(* CODESYS project M241_ILE_writeCSV.project
   Title: M241-ILS2K
   Version: 0.0.0.0
   Author: Philippe

Project tree, tasks and I/O mapping:
  MyController : TM241CE40R, Schneider Electric, order no. TM241CE40R, version 5.1.9.44
    application Application
      libraries: Integrated Lexium Library, 3.2.1.0 (Schneider Electric); FileFormatUtility, 1.5.15.0 (Schneider Electric)
      task MAST (cyclic, interval 20 ms, priority 15, watchdog 100 ms x 1) calls UPDATE_COMMAND, MAIN_SFC, CONSIGNE_VITESSE, ILE_functionblocks
      task Initialisation_IO (event, event StartApp, priority 1) calls nothing
      global variables GVL
      visualisation Visualization
      program ILE_functionblocks [FBD]
      program MAIN_SFC [SFC]
      visualisation Visualization_1
      program UPDATE_COMMAND [SFC]: WRITE_TABLE
      program CONSIGNE_VITESSE [ST]
    DI : Digital Inputs, Schneider Electric, version 5.1.9.44
        input  idwDI_IDW0 : DWORD  // IDW0
        input  ibDI_IB1 : BYTE  // IB1
    DQ : Digital Outputs, Schneider Electric, version 5.1.9.44
        output qwDQ_QW0 : WORD  // QW0
        output qbDQ_QB1 : BYTE  // QB1
    Counters : Counters, Schneider Electric, version 5.1.9.44
    Pulse_Generators : Pulse Generators, Schneider Electric, version 5.1.9.44
    Cartridge_1 : Cartridge, Schneider Electric, version 5.1.9.44
    Cartridge_2 : Cartridge, Schneider Electric, version 5.1.9.44
    IO_Bus : IO bus - TM3, Schneider Electric, version 5.1.9.44
    COM_Bus : COM bus, Schneider Electric, version 5.1.9.44
    Ethernet_1 : Ethernet Network, Schneider Electric, version 5.1.9.44
        settings: IPAddress = [192, 168, 100, 200]; SubnetMask = [255, 255, 255, 0]; GatewayAddress = [192, 168, 100, 254]; WebServer = TRUE; FTP Server = TRUE; SoMachine Protocol = TRUE; Modbus Server = TRUE; NetManage Protocol = TRUE; SNMP protocol = TRUE; Enable Routing = FALSE; WebVisu protocol = TRUE; DHCP Server Active = TRUE; Secured Web Server = TRUE
      Gestionnaire_Ethernet_Industriel : Industrial Ethernet Manager, Schneider Electric, version 1.0.12.40
          settings: BinaryFileSize = 586; Dhcps Host 0.Client Mac Address = [16#00, 16#80, 16#F4, 16#7B, 16#28, 16#E1]; Dhcps Host 0.Client Device Name = 'Lexium-ILx-002'; Dhcps Host 0.Client IP Address = [192, 168, 100, 159]; Dhcps Host 0.Network Mask = [255, 255, 255, 0]; Dhcps Host 0.Default Gateway = [192, 168, 100, 200]; Dhcps Host 2.Client Mac Address = [16#0, 16#0, 16#0, 16#0, 16#0]; Dhcps Host 3.Client Mac Address = [16#0, 16#0, 16#0, 16#0, 16#0]; Dhcps Host 4.Client Mac Address = [16#0, 16#0, 16#0, 16#0, 16#0]; Dhcps Host 5.Client Mac Address = [16#0, 16#0, 16#0, 16#0, 16#0]; Dhcps Host 6.Client Mac Address = [16#0, 16#0, 16#0, 16#0, 16#0]; Dhcps Host 7.Client Mac Address = [16#0, 16#0, 16#0, 16#0, 16#0]; Dhcps Host 8.Client Mac Address = [16#0, 16#0, 16#0, 16#0, 16#0]; Dhcps Host 9.Client Mac Address = [16#0, 16#0, 16#0, 16#0, 16#0]; Dhcps Host 10.Client Mac Address = [16#0, 16#0, 16#0, 16#0, 16#0]; Dhcps Host 11.Client Mac Address = [16#0, 16#0, 16#0, 16#0, 16#0]; Dhcps Host 12.Client Mac Address = [16#0, 16#0, 16#0, 16#0, 16#0]; Dhcps Host 13.Client Mac Address = [16#0, 16#0, 16#0, 16#0, 16#0]; Dhcps Host 14.Client Mac Address = [16#0, 16#0, 16#0, 16#0, 16#0]; Dhcps Host 15.Client Mac Address = [16#0, 16#0, 16#0, 16#0, 16#0]; Dhcps Host 16.Client Mac Address = [16#0, 16#0, 16#0, 16#0, 16#0]; Dhcps Host 17.Client Mac Address = [16#0, 16#0, 16#0, 16#0, 16#0]; Dhcps Host 18.Client Mac Address = [16#0, 16#0, 16#0, 16#0, 16#0]; Dhcps Host 19.Client Mac Address = [16#0, 16#0, 16#0, 16#0, 16#0]; Dhcps Host 20.Client Mac Address = [16#0, 16#0, 16#0, 16#0, 16#0]; Dhcps Host 21.Client Mac Address = [16#0, 16#0, 16#0, 16#0, 16#0]; Dhcps Host 22.Client Mac Address = [16#0, 16#0, 16#0, 16#0, 16#0]; Dhcps Host 23.Client Mac Address = [16#0, 16#0, 16#0, 16#0, 16#0]; Dhcps Host 24.Client Mac Address = [16#0, 16#0, 16#0, 16#0, 16#0]; Dhcps Host 25.Client Mac Address = [16#0, 16#0, 16#0, 16#0, 16#0]; Dhcps Host 26.Client Mac Address = [16#0, 16#0, 16#0, 16#0, 16#0]; Dhcps Host 27.Client Mac Address = [16#0, 16#0, 16#0, 16#0, 16#0]; Dhcps Host 28.Client Mac Address = [16#0, 16#0, 16#0, 16#0, 16#0]; Dhcps Host 29.Client Mac Address = [16#0, 16#0, 16#0, 16#0, 16#0]; Dhcps Host 30.Client Mac Address = [16#0, 16#0, 16#0, 16#0, 16#0]; Dhcps Host 31.Client Mac Address = [16#0, 16#0, 16#0, 16#0, 16#0]; Dhcps Host 32.Client Mac Address = [16#0, 16#0, 16#0, 16#0, 16#0]; Dhcps Host 33.Client Mac Address = [16#0, 16#0, 16#0, 16#0, 16#0]; Dhcps Host 34.Client Mac Address = [16#0, 16#0, 16#0, 16#0, 16#0]; Dhcps Host 35.Client Mac Address = [16#0, 16#0, 16#0, 16#0, 16#0];
            Dhcps Host 36.Client Mac Address = [16#0, 16#0, 16#0, 16#0, 16#0]; Dhcps Host 37.Client Mac Address = [16#0, 16#0, 16#0, 16#0, 16#0]; Dhcps Host 38.Client Mac Address = [16#0, 16#0, 16#0, 16#0, 16#0]; Dhcps Host 39.Client Mac Address = [16#0, 16#0, 16#0, 16#0, 16#0]; Dhcps Host 40.Client Mac Address = [16#0, 16#0, 16#0, 16#0, 16#0]; Dhcps Host 41.Client Mac Address = [16#0, 16#0, 16#0, 16#0, 16#0]; Dhcps Host 42.Client Mac Address = [16#0, 16#0, 16#0, 16#0, 16#0]; Dhcps Host 43.Client Mac Address = [16#0, 16#0, 16#0, 16#0, 16#0]; Dhcps Host 44.Client Mac Address = [16#0, 16#0, 16#0, 16#0, 16#0]; Dhcps Host 45.Client Mac Address = [16#0, 16#0, 16#0, 16#0, 16#0]; Dhcps Host 46.Client Mac Address = [16#0, 16#0, 16#0, 16#0, 16#0]; Dhcps Host 47.Client Mac Address = [16#0, 16#0, 16#0, 16#0, 16#0]; Dhcps Host 48.Client Mac Address = [16#0, 16#0, 16#0, 16#0, 16#0]; Dhcps Host 49.Client Mac Address = [16#0, 16#0, 16#0, 16#0, 16#0]; Dhcps Host 50.Client Mac Address = [16#0, 16#0, 16#0, 16#0, 16#0]; Dhcps Host 51.Client Mac Address = [16#0, 16#0, 16#0, 16#0, 16#0]; Dhcps Host 52.Client Mac Address = [16#0, 16#0, 16#0, 16#0, 16#0]; Dhcps Host 53.Client Mac Address = [16#0, 16#0, 16#0, 16#0, 16#0]; Dhcps Host 54.Client Mac Address = [16#0, 16#0, 16#0, 16#0, 16#0]; Dhcps Host 55.Client Mac Address = [16#0, 16#0, 16#0, 16#0, 16#0]; Dhcps Host 56.Client Mac Address = [16#0, 16#0, 16#0, 16#0, 16#0]; Dhcps Host 57.Client Mac Address = [16#0, 16#0, 16#0, 16#0, 16#0]; Dhcps Host 58.Client Mac Address = [16#0, 16#0, 16#0, 16#0, 16#0]; Dhcps Host 59.Client Mac Address = [16#0, 16#0, 16#0, 16#0, 16#0]; Dhcps Host 60.Client Mac Address = [16#0, 16#0, 16#0, 16#0, 16#0]; Dhcps Host 61.Client Mac Address = [16#0, 16#0, 16#0, 16#0, 16#0]; Dhcps Host 62.Client Mac Address = [16#0, 16#0, 16#0, 16#0, 16#0]; Dhcps Host 63.Client Mac Address = [16#0, 16#0, 16#0, 16#0, 16#0]; Dhcps Host 64.Client Mac Address = [16#0, 16#0, 16#0, 16#0, 16#0]; Dhcps Host 65.Client Mac Address = [16#0, 16#0, 16#0, 16#0, 16#0]; Dhcps Host 66.Client Mac Address = [16#0, 16#0, 16#0, 16#0, 16#0]; Dhcps Host 67.Client Mac Address = [16#0, 16#0, 16#0, 16#0, 16#0]; Dhcps Host 68.Client Mac Address = [16#0, 16#0, 16#0, 16#0, 16#0]; Dhcps Host 69.Client Mac Address = [16#0, 16#0, 16#0, 16#0, 16#0]; Dhcps Host 70.Client Mac Address = [16#0, 16#0, 16#0, 16#0, 16#0]; Dhcps Host 71.Client Mac Address = [16#0, 16#0, 16#0, 16#0, 16#0]; Dhcps Host 72.Client Mac Address = [16#0, 16#0, 16#0, 16#0, 16#0]; Dhcps Host 73.Client Mac Address = [16#0, 16#0, 16#0, 16#0, 16#0]; Dhcps Host 74.Client Mac Address = [16#0, 16#0, 16#0, 16#0, 16#0]; Dhcps Host 75.Client Mac Address = [16#0, 16#0, 16#0, 16#0, 16#0];
            Dhcps Host 76.Client Mac Address = [16#0, 16#0, 16#0, 16#0, 16#0]; Dhcps Host 77.Client Mac Address = [16#0, 16#0, 16#0, 16#0, 16#0]; Dhcps Host 78.Client Mac Address = [16#0, 16#0, 16#0, 16#0, 16#0]; Dhcps Host 79.Client Mac Address = [16#0, 16#0, 16#0, 16#0, 16#0]; Dhcps Host 80.Client Mac Address = [16#0, 16#0, 16#0, 16#0, 16#0]; Dhcps Host 81.Client Mac Address = [16#0, 16#0, 16#0, 16#0, 16#0]; Dhcps Host 82.Client Mac Address = [16#0, 16#0, 16#0, 16#0, 16#0]; Dhcps Host 83.Client Mac Address = [16#0, 16#0, 16#0, 16#0, 16#0]; Dhcps Host 84.Client Mac Address = [16#0, 16#0, 16#0, 16#0, 16#0]; Dhcps Host 85.Client Mac Address = [16#0, 16#0, 16#0, 16#0, 16#0]; Dhcps Host 86.Client Mac Address = [16#0, 16#0, 16#0, 16#0, 16#0]; Dhcps Host 87.Client Mac Address = [16#0, 16#0, 16#0, 16#0, 16#0]; Dhcps Host 88.Client Mac Address = [16#0, 16#0, 16#0, 16#0, 16#0]; Dhcps Host 89.Client Mac Address = [16#0, 16#0, 16#0, 16#0, 16#0]; Dhcps Host 90.Client Mac Address = [16#0, 16#0, 16#0, 16#0, 16#0]; Dhcps Host 91.Client Mac Address = [16#0, 16#0, 16#0, 16#0, 16#0]; Dhcps Host 92.Client Mac Address = [16#0, 16#0, 16#0, 16#0, 16#0]; Dhcps Host 93.Client Mac Address = [16#0, 16#0, 16#0, 16#0, 16#0]; Dhcps Host 94.Client Mac Address = [16#0, 16#0, 16#0, 16#0, 16#0]; Dhcps Host 95.Client Mac Address = [16#0, 16#0, 16#0, 16#0, 16#0]; Dhcps Host 96.Client Mac Address = [16#0, 16#0, 16#0, 16#0, 16#0]; Dhcps Host 97.Client Mac Address = [16#0, 16#0, 16#0, 16#0, 16#0]; Dhcps Host 98.Client Mac Address = [16#0, 16#0, 16#0, 16#0, 16#0]; Dhcps Host 99.Client Mac Address = [16#0, 16#0, 16#0, 16#0, 16#0]; Dhcps Host 100.Client Mac Address = [16#0, 16#0, 16#0, 16#0, 16#0]; Dhcps Host 101.Client Mac Address = [16#0, 16#0, 16#0, 16#0, 16#0]; Dhcps Host 102.Client Mac Address = [16#0, 16#0, 16#0, 16#0, 16#0]; Dhcps Host 103.Client Mac Address = [16#0, 16#0, 16#0, 16#0, 16#0]; Dhcps Host 104.Client Mac Address = [16#0, 16#0, 16#0, 16#0, 16#0]; Dhcps Host 105.Client Mac Address = [16#0, 16#0, 16#0, 16#0, 16#0]; Dhcps Host 106.Client Mac Address = [16#0, 16#0, 16#0, 16#0, 16#0]; Dhcps Host 107.Client Mac Address = [16#0, 16#0, 16#0, 16#0, 16#0]; Dhcps Host 108.Client Mac Address = [16#0, 16#0, 16#0, 16#0, 16#0]; Dhcps Host 109.Client Mac Address = [16#0, 16#0, 16#0, 16#0, 16#0]; Dhcps Host 110.Client Mac Address = [16#0, 16#0, 16#0, 16#0, 16#0]; Dhcps Host 111.Client Mac Address = [16#0, 16#0, 16#0, 16#0, 16#0]; Dhcps Host 112.Client Mac Address = [16#0, 16#0, 16#0, 16#0, 16#0]; Dhcps Host 113.Client Mac Address = [16#0, 16#0, 16#0, 16#0, 16#0]; Dhcps Host 114.Client Mac Address = [16#0, 16#0, 16#0, 16#0, 16#0]; Dhcps Host 115.Client Mac Address = [16#0, 16#0, 16#0, 16#0, 16#0];
            Dhcps Host 116.Client Mac Address = [16#0, 16#0, 16#0, 16#0, 16#0]; Dhcps Host 117.Client Mac Address = [16#0, 16#0, 16#0, 16#0, 16#0]; Dhcps Host 118.Client Mac Address = [16#0, 16#0, 16#0, 16#0, 16#0]; Dhcps Host 119.Client Mac Address = [16#0, 16#0, 16#0, 16#0, 16#0]; Dhcps Host 120.Client Mac Address = [16#0, 16#0, 16#0, 16#0, 16#0]; Dhcps Host 121.Client Mac Address = [16#0, 16#0, 16#0, 16#0, 16#0]; Dhcps Host 122.Client Mac Address = [16#0, 16#0, 16#0, 16#0, 16#0]; Dhcps Host 123.Client Mac Address = [16#0, 16#0, 16#0, 16#0, 16#0]; Dhcps Host 124.Client Mac Address = [16#0, 16#0, 16#0, 16#0, 16#0]; Dhcps Host 125.Client Mac Address = [16#0, 16#0, 16#0, 16#0, 16#0]; Dhcps Host 126.Client Mac Address = [16#0, 16#0, 16#0, 16#0, 16#0]; Dhcps Host 127.Client Mac Address = [16#0, 16#0, 16#0, 16#0, 16#0]; Dhcps Host 128.Client Mac Address = [16#0, 16#0, 16#0, 16#0, 16#0]; serialized Values = 010bc991-f7f9-45b2-8b15-1d199ae18604=0|; InterfaceUsedByDhcpSize = 4; InterfaceUsedByDhcp = [192,168,100,200]
          unmapped channels: Global Status, Healthbit 0, Healthbit 1, Healthbit 2, Healthbit 3, Channels 0, Channels 1, Channels 2, Channels 3
        Lexium_ILE : Lexium ILE, Schneider Electric, order no. 89330, version 1.2.11.0
            settings: IP address of Target = [192,168,100,159]; MAC address of Target = [16#00, 16#80, 16#F4, 16#7B, 16#28, 16#E1]; DeviceNumber = 1; Object Input1 = [0, 40, 268500992, 257]; Object Output1 = [1, 40, 268566528, 257]; Connection Id List = [257,0,0,0,0,0,0,0]; Connection Settings.Connection Number = 257
            unmapped channels: Input Read/Write IclA, Output Read/Write IclA
    Serial_Line_1 : Serial line, Schneider Electric, version 5.1.9.44
      SoMachine_Network_Manager : Machine Expert-Network Manager, Schneider Electric, version 4.0.0.4
    Serial_Line_2 : Serial line, Schneider Electric, version 5.1.9.44
      Modbus_Manager : Modbus Manager, Schneider Electric, version 4.0.0.4
  libraries: VisuSymbols, 3.5.10.0 (System)
  text list GlobalTextList
*)

// MyController/Application/GVL

VAR_GLOBAL
	
	// Power
	ILE_Power_Enable : BOOL := FALSE;
	ILE_Power_StatusOK: BOOL;
	
	// LimitSwitches
	ILE_LimitSwitch_Execute : BOOL;
	ILE_LimitSwitch_neg_disabled,ILE_LimitSwitch_pos_disabled : BOOL;
	 
	// Movement (target velocity)
 	ILE_Movement : BOOL;
 	targetVelocity : DINT := 0;
	actualVelocity : DINT;
	inVelocity : BOOL;
	
	// Error reading
	ILE_ReadError : BOOL := TRUE;
	ILE_ReadStatus : BOOL := TRUE;
	ILE_ReadPosition : BOOL := TRUE;
	
	ILE_Reset : BOOL;
	ILE_ResetOK : BOOL;
	
	StartApp : BOOL;
	
	// Array to output data
  
	csvWrite :FFU.FB_CsvWrite;  
	// xCmdWrite :BOOL;  
	tableLogData:ARRAY[0..csv_NumOfRows-1,0..csv_NumOfColumns-  1] OF STRING(csv_LengthOfValue);  
	csvTable: FFU.ST_CsvTable;  

END_VAR

VAR_GLOBAL CONSTANT
	
	// CVS table size
	csv_NumOfRows :UINT:= 3000;  
	csv_NumOfColumns :UINT:= 2; // i et actual vel  
	csv_LengthOfValue :UINT:= 30;
	
END_VAR

// MyController/Application/UPDATE_COMMAND
PROGRAM UPDATE_COMMAND
VAR
END_VAR

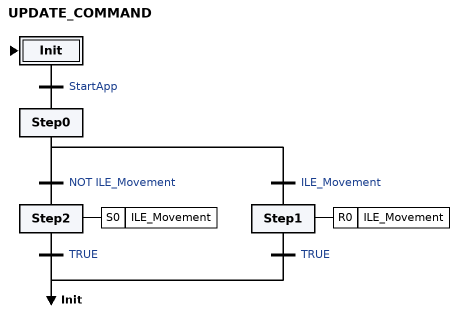
INITIAL_STEP Init:
END_STEP
TRANSITION FROM Init TO Step0
    := StartApp;
END_TRANSITION
STEP Step0:
END_STEP
TRANSITION FROM Step0 TO Step2
    := NOT ILE_Movement;
END_TRANSITION
STEP Step2:
    ILE_Movement(S0);
END_STEP
TRANSITION FROM Step2 TO Init
    := TRUE;
END_TRANSITION
TRANSITION FROM Step0 TO Step1
    := ILE_Movement;
END_TRANSITION
STEP Step1:
    ILE_Movement(R0);
END_STEP
TRANSITION FROM Step1 TO Init
    := TRUE;
END_TRANSITION

ACTION WRITE_TABLE:

END_ACTION

END_PROGRAM

// MyController/Application/MAIN_SFC
PROGRAM MAIN_SFC
VAR
	ILE_ManualStart: BOOL;
END_VAR

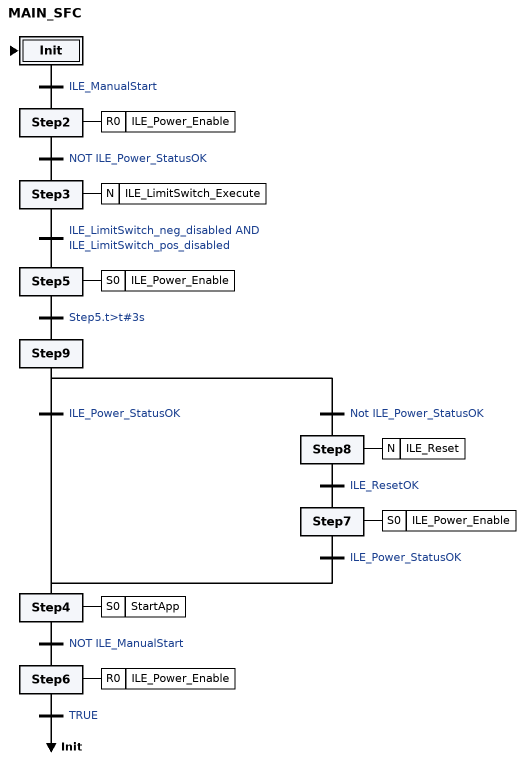
INITIAL_STEP Init:
END_STEP
TRANSITION FROM Init TO Step2
    := ILE_ManualStart;
END_TRANSITION
STEP Step2:
    ILE_Power_Enable(R0);
END_STEP
TRANSITION FROM Step2 TO Step3
    := NOT ILE_Power_StatusOK;
END_TRANSITION
STEP Step3:
    ILE_LimitSwitch_Execute(N);
END_STEP
TRANSITION FROM Step3 TO Step5
    := ILE_LimitSwitch_neg_disabled AND ILE_LimitSwitch_pos_disabled;
END_TRANSITION
STEP Step5:
    ILE_Power_Enable(S0);
END_STEP
TRANSITION FROM Step5 TO Step9
    := Step5.t>t#3s;
END_TRANSITION
STEP Step9:
END_STEP
TRANSITION FROM Step9 TO Step4
    := ILE_Power_StatusOK;
END_TRANSITION
TRANSITION FROM Step9 TO Step8
    := Not ILE_Power_StatusOK;
END_TRANSITION
STEP Step8:
    ILE_Reset(N);
END_STEP
TRANSITION FROM Step8 TO Step7
    := ILE_ResetOK;
END_TRANSITION
STEP Step7:
    ILE_Power_Enable(S0);
END_STEP
TRANSITION FROM Step7 TO Step4
    := ILE_Power_StatusOK;
END_TRANSITION
STEP Step4:
    StartApp(S0);
END_STEP
TRANSITION FROM Step4 TO Step6
    := NOT ILE_ManualStart;
END_TRANSITION
STEP Step6:
    ILE_Power_Enable(R0);
END_STEP
TRANSITION FROM Step6 TO Init
    := TRUE;
END_TRANSITION

END_PROGRAM

// MyController/Application/CONSIGNE_VITESSE
PROGRAM CONSIGNE_VITESSE

VAR CONSTANT
	
	vmax : REAL := 1000.0;
	nbStepAcc : DINT := 250;
	nbStepRun : DINT := 500;
	nbStepDecc : DINT := 250;

END_VAR


VAR
	nbTotalStep : DINT;
	i : DINT := 0;
	j : DINT := 0;
END_VAR

nbTotalStep := nbStepAcc + nbStepRun + nbStepDecc;
i := (i+1) MOD nbTotalStep;

IF i <= nbStepAcc THEN
	targetVelocity :=  REAL_TO_INT(vmax * DINT_TO_REAL(i/nbStepAcc));
ELSIF i <= nbStepAcc + nbStepRun THEN
	targetVelocity  :=  REAL_TO_INT(vmax);
ELSE
	targetVelocity := REAL_TO_INT( vmax * (1.0 - DINT_TO_REAL( (i - (nbStepAcc + nbStepRun)) )/ DINT_TO_REAL(nbStepDecc)) );
END_IF

// writing data in table

j := j+1;
IF j < csv_NumOfRows THEN
	// writing data in table
	tableLogData [j,0] := DINT_TO_STRING(j);
	tableLogData [j,1] := DINT_TO_STRING(actualVelocity);
ELSIF j = csv_NumOfRows THEN
	// writing table in CVS file
	csvWrite.i_stTableWriteValues.pbyTable := ADR(tableLogData);  
	csvWrite.i_stTableWriteValues.uiNumOfRows := csv_NumOfRows;  
	csvWrite.i_stTableWriteValues.uiNumOfColumns := csv_NumOfColumns;
	csvWrite.i_stTableWriteValues.udiSizeOfTable := SIZEOF(tableLogData);  
	csvWrite.i_stWriteParameter.sDelimiter := ';';  
	csvWrite.i_stWriteParameter.etModeFileOpen := FFU.ET_ModeFileOpen.Append;  
//	csvWrite.i_stWriteParameter.uiNumOfRows := 3;  
//	csvWrite.i_stWriteParameter.uiNumOfColumns := csv_NumOfColumns;  
	csvWrite(  
		i_xExecute:= TRUE,  
		i_sFilePath:= '/sd0/actual_velocity.csv',  
		i_stWriteParameter:= ,  
		i_timTimeout:= ,  
		i_stTableWriteValues:= ,  
		q_xDone=> ,  
		q_xBusy=> ,  
		q_xError=> ,  
		q_etResult=> ,  
		q_sResultMsg=> ,  
		q_udiFileSize=> );
	
END_IF

END_PROGRAM

// MyController/Application/ILE_functionblocks
PROGRAM ILE_functionblocks
VAR
	MC_Power: GIPLC.MC_Power;;
	MC_ReadAxisError: GIPLC.MC_ReadAxisError;
	SetLimitSwitch_ILX_pos : GILXM.SetLimitSwitch_ILX;
	SetLimitSwitch_ILX_neg : GILXM.SetLimitSwitch_ILX;
	MC_ReadActualPosition: GIPLC.MC_ReadActualPosition;
	MC_ReadStatus: GIPLC.MC_ReadStatus;
	
	MC_MoveVelocity: GIPLC.MC_MoveVelocity;
	MC_Reset: GIPLC.MC_Reset;
	MC_ReadActualVelocity: GIPLC.MC_ReadActualVelocity;
END_VAR

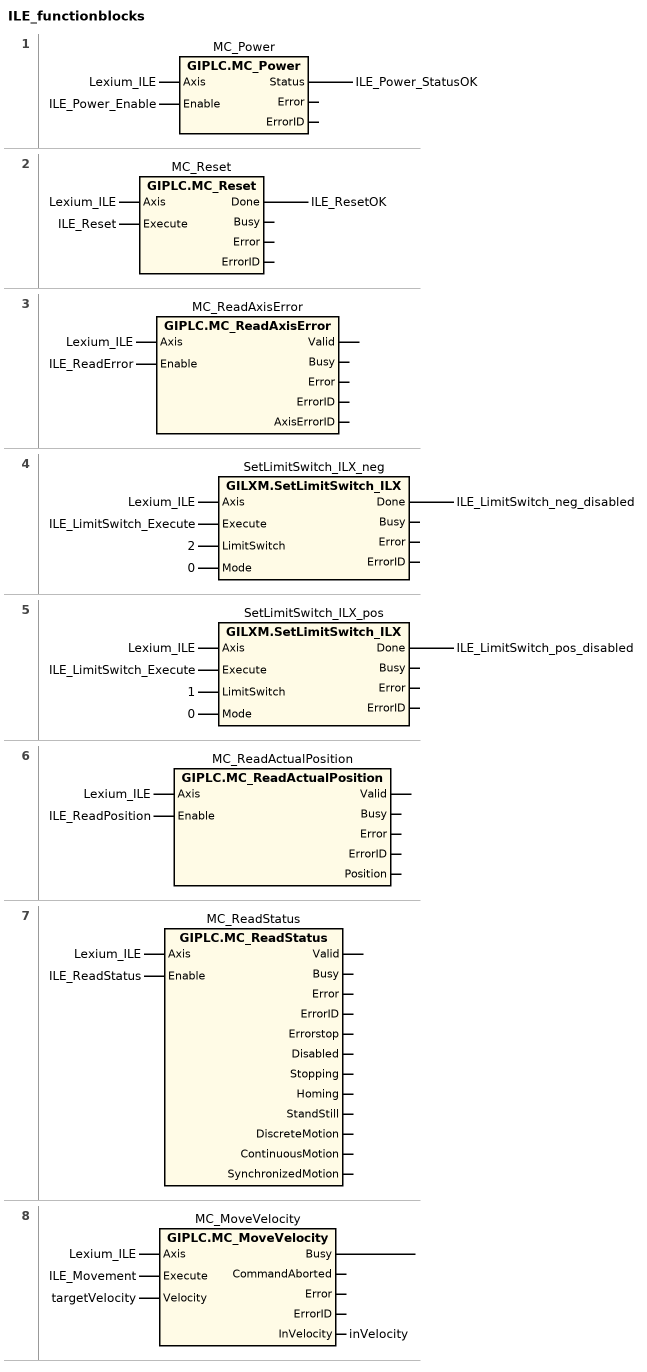
// NETWORK 1
MC_Power(Axis := Lexium_ILE, Enable := ILE_Power_Enable); // GIPLC.MC_Power
ILE_Power_StatusOK := MC_Power.Status;

// NETWORK 2
MC_Reset(Axis := Lexium_ILE, Execute := ILE_Reset); // GIPLC.MC_Reset
ILE_ResetOK := MC_Reset.Done;

// NETWORK 3
MC_ReadAxisError(Axis := Lexium_ILE, Enable := ILE_ReadError); // GIPLC.MC_ReadAxisError

// NETWORK 4
SetLimitSwitch_ILX_neg(Axis := Lexium_ILE, Execute := ILE_LimitSwitch_Execute, LimitSwitch := 2, Mode := 0); // GILXM.SetLimitSwitch_ILX
ILE_LimitSwitch_neg_disabled := SetLimitSwitch_ILX_neg.Done;

// NETWORK 5
SetLimitSwitch_ILX_pos(Axis := Lexium_ILE, Execute := ILE_LimitSwitch_Execute, LimitSwitch := 1, Mode := 0); // GILXM.SetLimitSwitch_ILX
ILE_LimitSwitch_pos_disabled := SetLimitSwitch_ILX_pos.Done;

// NETWORK 6
MC_ReadActualPosition(Axis := Lexium_ILE, Enable := ILE_ReadPosition); // GIPLC.MC_ReadActualPosition

// NETWORK 7
MC_ReadStatus(Axis := Lexium_ILE, Enable := ILE_ReadStatus); // GIPLC.MC_ReadStatus

// NETWORK 8
MC_MoveVelocity(
    Axis := Lexium_ILE,
    Execute := ILE_Movement,
    Velocity := targetVelocity,
    InVelocity => inVelocity); // GIPLC.MC_MoveVelocity

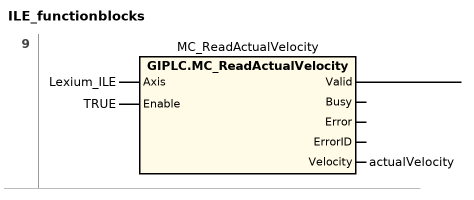
// NETWORK 9
MC_ReadActualVelocity(Axis := Lexium_ILE, Enable := TRUE, Velocity => actualVelocity); // GIPLC.MC_ReadActualVelocity

END_PROGRAM

// MyController/Application/Visualization
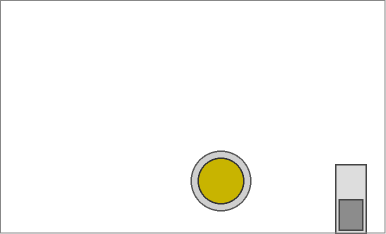
VISUALIZATION Visualization  // 386x234
    Lamp1 (186,146 70x70), variable: ILE_functionblocks.power, style: Lamp-Lamp1-Yellow
    DipSwitch (316,164 70x70), behaviour: TOGGLE, style: Switch-DipSwitch-Gray
END_VISUALIZATION

// MyController/Application/Visualization_1
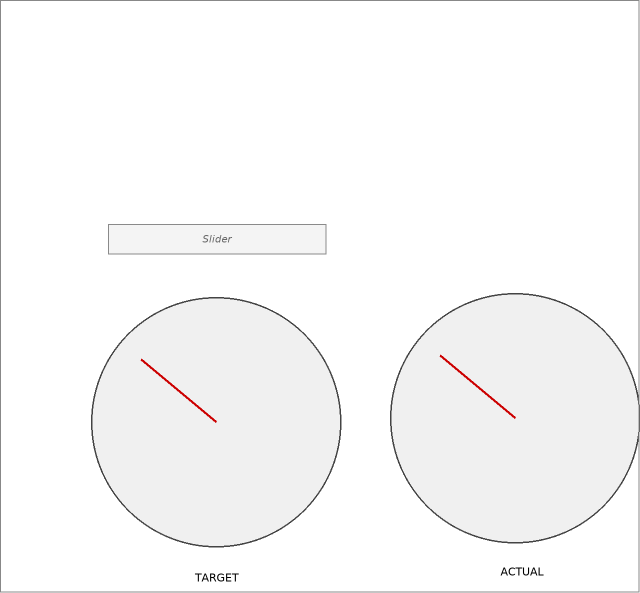
VISUALIZATION Visualization_1  // 640x593
    Slider (108,224 218x30), variable: targetVelocity, scale 0..4900
    Meter360 (390,293 250x250), value: actualVelocity, style: Meter-Meter360-Gray, scale format: %.1f, scale 0..5000
    Meter360 (91,297 250x250), value: targetVelocity, style: Meter-Meter360-Gray, scale format: %.1f, scale 0..5000
    Label (142,563 150x30), "TARGET"
    Label (447,557 150x30), "ACTUAL"
END_VISUALIZATION
